// Mitsubishi GX Works2 project: 乙級第三題-ST   PLC: FX3U/FX3UC

// task Task_01 (event TRUE, interval 0, priority 31): POU_01

PROGRAM POU_01
VAR
  wProgramStep : INT;
  wPulse : INT;
  wSpeed : INT;
  tdT143 : TON;
  tdT201 : TON;
  tdT202 : TON;
  bM0 : BOOL;
  bServoRun : BOOL;
  bServoRev : BOOL;
  bM143 : BOOL;
  bM133 : BOOL;
  bM17 : BOOL;
  tdT200 : TON;
  tdT144 : TON;
  tdT203 : TON;
  bStarted : BOOL;
  tdTX11 : TON;
  trigX11 : F_TRIG;
  tdT50 : TON;
  tdT21 : TON;
  tdT60 : TON;
  tdT61 : TON;
  tdT70 : TON;
  tdT73 : TON;
  tdT62 : TON;
  tdT43 : TON;
  tdT71 : TON;
  tdT75 : TON;
  tdT42 : TON;
  tdT72 : TON;
  tdT22 : TON;
  tdT24 : TON;
  tdT27 : TON;
  tdT28 : TON;
END_VAR
VAR CONSTANT
  W_ORG_POS : INT := 16100;
  W_FRONT_INSTALL_POS : INT := 13600;
END_VAR
VAR
  tdT30 : TON;
  tdT31 : TON;
  tdT33 : TON;
  tdT35 : TON;
  tdT25 : TON;
  tdT36 : TON;
  bJawClosed : BOOL;
  bReachOrg : BOOL;
END_VAR
VAR CONSTANT
  W_REAR_INSTALL_POS : INT := 9600;
END_VAR
(* 機電整合乙級術科第三題
   Author: Steven Luo
   Date: 2018/10/25
*)

IF M8000 THEN
	Y17 := TRUE;
END_IF;

IF M8002 THEN
	D8342 := 3000;
	D8343 := 10000;
	D8348 := 1000;
	D8349 := 1000;
	bServoRun := FALSE;
	bServoRev := FALSE;
	bM0 := FALSE;
	bM17 := FALSE;
	bM143 := FALSE;
	tdT200(IN := FALSE);
	wProgramStep := 0;
END_IF;

IF M133 THEN
	bM133 := TRUE;
END_IF;

IF Y11 THEN
	bJawClosed := TRUE;
ELSE
	bJawClosed := FALSE;
END_IF;

IF NOT M144 AND NOT bM17 THEN
	IF bM0 THEN
		D5 := 0;
	ELSE
		D5 := 310;
	END_IF;
END_IF;

IF NOT X17 THEN (* 急停 *)
	ZRST(TRUE, Y0, Y10);
	ZRST(TRUE, Y13, Y16);
(*	M8349 := TRUE;*)
	bServoRun := FALSE;
	D5 := 313;
	bStarted := FALSE;
	bM17 := TRUE;
	M144 := FALSE;
	tdT201(IN := FALSE);
	tdT202(IN := FALSE);
	tdT203(IN := FALSE);
	wProgramStep := -1;
END_IF;

IF X17 AND bM17 AND M136 THEN
	D5 := 312;
(*	M8349 := FALSE;*)
	IF M132 THEN (* 解除急停，按下復歸 *)
		bM17 := FALSE;
		bM143 := TRUE;
		tdT143(IN := FALSE);
		tdT144(IN := FALSE);
		wProgramStep := 201;
	END_IF;
END_IF;

IF bM143 THEN (* 黃燈閃爍 *)
	tdT143(IN := NOT tdT144.Q, PT := T#500ms);
	tdT144(IN := tdT143.Q, PT := T#500ms);
	M143 := tdT143.Q;
END_IF;

IF X3 AND X6 AND NOT Y13 AND NOT Y14 AND NOT Y15 AND NOT Y16 AND NOT M136 THEN
	IF D8140 = W_ORG_POS THEN 
		bM0 := TRUE; (* 原點條件 *)
	END_IF;
ELSE
	bM0 := FALSE;
END_IF;

PLSR(bServoRun, wSpeed, wPulse, D8349, Y0);
OUT(bServoRev, Y4);

D4 := D1 + D2 + D3;

CASE wProgramStep OF
0:
	IF X17 THEN
		IF M130 THEN
			tdT201(IN := FALSE);
			tdT202(IN := FALSE);
			tdT203(IN := FALSE);
			wProgramStep := 200;
		ELSE
			wProgramStep := 20;
		END_IF;
	END_IF;
20:
	IF M130 THEN
		wProgramStep := 0;
	END_IF;
	IF bM0 THEN
		ZRST(TRUE, D0, D5);
		ZRST(TRUE, M150, M152);
		ZRST(TRUE, M160, M164);
		bM133 := FALSE;
		bM143 := FALSE;
		bReachOrg := FALSE;
		M142 := TRUE;
		M143 := FALSE;
		M144 := FALSE;
		tdT21(IN := FALSE);
		tdT22(IN := FALSE);
		tdT24(IN := FALSE);
		tdT25(IN := FALSE);
		tdT27(IN := FALSE);
		tdT28(IN := FALSE);
		tdT30(IN := FALSE);
		tdT31(IN := FALSE);
		tdT33(IN := FALSE);
		tdT35(IN := FALSE);
		tdT36(IN := FALSE);
		tdT42(IN := FALSE);
		tdT43(IN := FALSE);
		tdT50(IN := FALSE);
		tdT60(IN := FALSE);
		tdT61(IN := FALSE);
		tdT62(IN := FALSE);
		tdT70(IN := FALSE);
		tdT71(IN := FALSE);
		tdT72(IN := FALSE);
		tdT73(IN := FALSE);
		tdT75(IN := FALSE);
		tdTX11(IN := FALSE);
		IF M131 THEN
			bStarted := TRUE;
			M142 := FALSE;
			M144 := TRUE;
			wProgramStep := 21;
		END_IF;
	END_IF;
21:
	Y14 := TRUE; (* F輸送帶運轉 *)
	Y15 := TRUE; (* 定位缸 *)
	tdT21(IN := TRUE, PT := T#3s);
	IF tdT21.Q THEN
		Y14 := FALSE;
		Y15 := FALSE;
		wProgramStep := 20;
	END_IF;
	tdTX11(IN := TRUE, PT := T#2s);
	IF X11 THEN
		D20 := TIME_TO_INT(tdTX11.ET);
		ZCP(TRUE, 900, 1300, TIME_TO_INT(tdTX11.ET), M150);
		INCP(TRUE, D0);
	END_IF;
	trigX11(_CLK := X11);
	IF trigX11.Q THEN
		IF M150 THEN (* 凹槽朝前 *)
			wProgramStep := 60;
		ELSIF M151 THEN (* 凹槽朝後 *)
			wProgramStep := 60;
		ELSIF M152 THEN (* 凹槽朝下 *)
			wProgramStep := 50;
		END_IF;
	END_IF;
22: (* 組裝料組裝行程 *)
	Y15 := FALSE; (* 進料缸 *)
	Y6 := TRUE; (* B-水平缸縮回 *)
	IF X3 THEN (* Y軸氣壓缸後位 *)
		Y6 := FALSE;
		wProgramStep := 23;
	END_IF;
23:
	Y7 := TRUE; (* C+垂直缸下降 *)
	IF X7 THEN (* Z軸氣壓缸下位 *)
		Y7 := FALSE;
		wProgramStep := 24;
	END_IF;
24:
	tdT24(IN := TRUE, PT := T#500ms);
	IF tdT24.Q THEN
		wProgramStep := 25;
	END_IF;
25:
	Y11 := FALSE;
	Y12 := TRUE; (* D-夾爪放 *)
	tdT25(IN := TRUE, PT := T#500ms);
	IF tdT25.Q THEN
		Y12 := FALSE;
		IF M150 THEN
			M160 := FALSE;
		ELSIF M151 THEN
			M161 := FALSE;
		END_IF;
		wProgramStep := 26;
	END_IF;
26:
	Y10 := TRUE; (* C-垂直缸上升 *)
	IF X6 THEN (* Z軸氣壓缸上位 *)
		Y10 := FALSE;
		wProgramStep := 27;
	END_IF;
27:
	Y13 := TRUE; (* E分離缸分離 *)
	tdT27(IN := TRUE, PT := T#1000ms);
	IF tdT27.Q THEN
		Y13 := FALSE;
		wProgramStep := 28;
	END_IF;
28:
	IF X10 THEN
		D5 := 310;
		wPulse := W_FRONT_INSTALL_POS;
		bServoRun := TRUE;
		bServoRev := TRUE;
		tdT28(IN := TRUE, PT := T#500ms);
		IF NOT M8340 AND tdT28.Q THEN
			bServoRun := FALSE;
			bServoRev := FALSE;
			wProgramStep := 29;
		END_IF;
	ELSE
		D5 := 311;
	END_IF;
29:
	Y7 := TRUE; (* C+垂直缸下降 *)
	IF X7 THEN (* Z軸氣壓缸下位 *)
		Y7 := FALSE;
		wProgramStep := 30;
	END_IF;
30:
	tdT30(IN := TRUE, PT := T#500ms);
	IF tdT30.Q THEN
		wProgramStep := 31;
	END_IF;
31:
	Y11 := TRUE; (* D+夾爪夾 *)
	tdT31(IN := TRUE, PT := T#500ms);
	IF tdT31.Q THEN
		M162 := TRUE; (* 圓料夾取 *)
		wProgramStep := 32;
	END_IF;
32:
	Y10 := TRUE; (* C-垂直缸上升 *)
	IF X6 THEN (* Z軸氣壓缸上位 *)
		Y10 := FALSE;
		wProgramStep := 33;
	END_IF;
33:
	wPulse := W_FRONT_INSTALL_POS;
	bServoRun := TRUE;
	tdT33(IN := TRUE, PT := T#500ms);
	IF NOT M8340 AND tdT33.Q THEN
		bServoRun := FALSE;
		wProgramStep := 34;
	END_IF;
34:
	Y7 := TRUE; (* C+垂直缸下降 *)
	IF X7 THEN (* Z軸氣壓缸下位 *)
		Y7 := FALSE;
		wProgramStep := 35;
	END_IF;
35:
	Y11 := FALSE;
	Y12 := TRUE; (* D-夾爪放 *)
	tdT35(IN := TRUE, PT := T#500ms);
	IF tdT35.Q THEN
		Y12 := FALSE;
		M162 := FALSE;
		wProgramStep := 36;
	END_IF;
36:
	Y11 := TRUE; (* D+夾爪夾 *)
	tdT36(IN := TRUE, PT := T#500ms);
	IF tdT36.Q THEN
		IF M150 THEN
			M163 := TRUE; (* 凹槽朝前組裝 *)
		ELSIF M151 THEN
			M164 := TRUE; (* 凹槽朝後組裝 *)
		END_IF;
		wProgramStep := 37;
	END_IF;
37: (* 組裝料出料行程 *)
	Y10 := TRUE; (* C-垂直缸上升 *)
	IF X6 THEN (* Z軸氣壓缸上位 *)
		Y10 := FALSE;
		D1 := D1 + 1;
		wProgramStep := 70;
	END_IF;
40:
	Y5 := TRUE; (* B+水平缸伸出 *)
	IF X5 THEN (* Y軸氣壓缸前位 *)
		Y5 := FALSE;
		wProgramStep := 41;
	END_IF;
41:
	Y7 := TRUE; (* C+垂直缸下降 *)
	IF X7 THEN (* Z軸氣壓缸下位 *)
		Y7 := FALSE;
		wProgramStep := 42;
	END_IF;
42:
	tdT42(IN := TRUE, PT := T#500ms);
	IF tdT42.Q THEN
		wProgramStep := 43;
	END_IF;
43:
	Y11 := TRUE; (* D+夾爪夾 *)
	tdT43(IN := TRUE, PT := T#500ms);
	IF tdT43.Q THEN
		IF M150 THEN
			M160 := TRUE;
		ELSIF M151 THEN
			M161 := TRUE;
		END_IF;
		wProgramStep := 44;
	END_IF;
44:
	Y10 := TRUE; (* C-垂直缸上升 *)
	IF X6 THEN (* Z軸氣壓缸上位 *)
		Y10 := FALSE;
		IF M150 THEN
			wProgramStep := 22;
		ELSE
			wProgramStep := 45;
		END_IF;
	END_IF;
45: (* 非組裝料出料行程 *)
	Y6 := TRUE; (* B-水平缸縮回 *)
	IF X4 THEN (* Y軸氣壓缸中位 *)
		Y6 := FALSE;
		D2 := D2 + 1;;
		wProgramStep := 70;
	END_IF;
50: (* 反面出料行程 *)
	Y16 := TRUE; (* H定位缸 *)
	tdT50(IN := TRUE, PT := T#2500ms);
	IF tdT50.Q THEN
		Y16 := FALSE;
		D3 := D3 + 1;
		wProgramStep := 60;
	END_IF;
60:
	tdT60(IN := TRUE, PT := T#2500ms);
	IF tdT60.Q THEN
		Y14 := FALSE; (* F輸送帶停止 *)
		IF M150 THEN
			wProgramStep := 40;
		ELSE
			wProgramStep := 61;
		END_IF;
	END_IF;
61:
	tdT61(IN := TRUE, PT := T#500ms);
	IF tdT61.Q THEN
		wProgramStep := 62;
	END_IF;
62:
	Y15 := FALSE; (* 進料缸 *)
	tdT62(IN := TRUE, PT := T#500ms);
	IF tdT62.Q THEN
		IF M151 THEN
			wProgramStep := 40;
		ELSE
			IF NOT bM133 THEN
				tdT21(IN := FALSE);
				tdT22(IN := FALSE);
				tdT24(IN := FALSE);
				tdT25(IN := FALSE);
				tdT27(IN := FALSE);
				tdT28(IN := FALSE);
				tdT30(IN := FALSE);
				tdT31(IN := FALSE);
				tdT33(IN := FALSE);
				tdT35(IN := FALSE);
				tdT36(IN := FALSE);
				tdT42(IN := FALSE);
				tdT43(IN := FALSE);
				tdT50(IN := FALSE);
				tdT60(IN := FALSE);
				tdT61(IN := FALSE);
				tdT62(IN := FALSE);
				tdT70(IN := FALSE);
				tdT71(IN := FALSE);
				tdT72(IN := FALSE);
				tdT73(IN := FALSE);
				tdT75(IN := FALSE);
				tdTX11(IN := FALSE);
				wProgramStep := 21;
			ELSE
				wProgramStep := 0;
			END_IF;
		END_IF;
	END_IF;
70: (* 排料 *)
	wPulse := W_ORG_POS;
	wSpeed := D8343;
	bServoRun := TRUE;
	tdT70(IN := TRUE, PT := T#500ms);
	IF NOT M8340 AND tdT70.Q THEN
		bServoRun := FALSE;
		bReachOrg := TRUE;
		D8140 := 0;
		Y3 := TRUE; (* Servo CCLR *)
		tdT71(IN := TRUE, PT := T#500ms);
		IF tdT71.Q THEN
			Y3 := FALSE;
			wProgramStep := 71;
		END_IF;
	END_IF;
71:
	Y7 := TRUE; (* C+垂直缸下降 *)
	IF X7 THEN (* Z軸氣壓缸下位 *)
		Y7 := FALSE;
		IF M162 THEN
			wProgramStep := 73;
		ELSE
			wProgramStep := 72;
		END_IF;
	END_IF;
72:
	tdT72(IN := TRUE, PT := T#500ms);
	IF tdT72.Q THEN
		wProgramStep := 73;
	END_IF;
73:
	Y11 := FALSE;
	Y12 := TRUE; (* D-夾爪放 *)
	tdT73(IN := TRUE, PT := T#500ms);
	IF tdT73.Q THEN
		Y12 := FALSE;
		wProgramStep := 74;
	END_IF;
74:
	Y10 := TRUE; (* C-垂直缸上升 *)
	IF X6 THEN (* Z軸氣壓缸上位 *)
		Y10 := FALSE;
		wProgramStep := 75;
	END_IF;
75:
	wPulse := W_ORG_POS;
	bServoRun := TRUE;
	bServoRev := TRUE;
	tdT75(IN := TRUE, PT := T#500ms);
	IF NOT M8340 AND tdT75.Q THEN
		bServoRun := FALSE;
		bServoRev := FALSE;
		wProgramStep := 76;
	END_IF;
76:
	Y6 := TRUE; (* B-水平缸縮回 *)
	IF X3 THEN (* Y軸氣壓缸後位 *)
		Y6 := FALSE;
		IF NOT bM133 AND NOT bM143 THEN
			tdT21(IN := FALSE);
			tdT22(IN := FALSE);
			tdT24(IN := FALSE);
			tdT25(IN := FALSE);
			tdT27(IN := FALSE);
			tdT28(IN := FALSE);
			tdT30(IN := FALSE);
			tdT31(IN := FALSE);
			tdT33(IN := FALSE);
			tdT35(IN := FALSE);
			tdT36(IN := FALSE);
			tdT42(IN := FALSE);
			tdT43(IN := FALSE);
			tdT50(IN := FALSE);
			tdT60(IN := FALSE);
			tdT61(IN := FALSE);
			tdT62(IN := FALSE);
			tdT70(IN := FALSE);
			tdT71(IN := FALSE);
			tdT72(IN := FALSE);
			tdT73(IN := FALSE);
			tdT75(IN := FALSE);
			tdTX11(IN := FALSE);
			wProgramStep := 21;
		ELSE
			wProgramStep := 0;
		END_IF;
	END_IF;
100:
	Y5 := TRUE; (* B+水平缸伸出 *)
	IF X5 THEN (* Y軸氣壓缸前位 *)
		Y5 := FALSE;
		wProgramStep := 71;
	END_IF;
101:
	Y6 := TRUE; (* B-水平缸縮回 *)
	IF X3 THEN (* Y軸氣壓缸後位 *)
		Y6 := FALSE;
		wProgramStep := 102;
	END_IF;
102:
	Y5 := TRUE; (* B+水平缸伸出 *)
	IF X4 THEN (* Y軸氣壓缸中位 *)
		Y5 := FALSE;
		wProgramStep := 71;
	END_IF;
200:
	IF X6 THEN (* c0 Z軸上位 *)
		IF X3 THEN (* b0 Y軸後位 *)
			wSpeed := D8343;
			wPulse := 3000;
			OUT((NOT X0 AND M110) OR M111, bServoRun);
			OUT(M111 AND NOT M110, bServoRev);
			IF X0 THEN
				D8140 := 0;
				Y3 := TRUE; (* Servo CCLR *)
				tdT200(IN := TRUE, PT := T#500ms);
				IF tdT200.Q THEN
					Y3 := FALSE;
				END_IF;
			ELSE
				tdT200(IN := FALSE);
			END_IF;
		END_IF;
		OUT(M112, Y5); (* B+水平缸伸出 *)
		OUT(M113, Y6); (* B-水平缸縮回 *)
	END_IF;
	OUT(M114, Y10); (* C-垂直缸上升 *)
	OUT(M115, Y7); (* C+垂直缸下降 *)
	OUT(M116, Y11); (* D+夾爪夾 *)
	OUT(M117, Y12); (* D-夾爪放 *)
	OUT(M119, Y14); (* F輸送帶運轉 *)
	OUT(M118, Y13); (* E分離缸分離 *)
	OUT(M120, Y15); (* G進料缸進料 *)
	OUT(M121, Y16); (* H定位缸 *)
	IF M137 OR M132 THEN (* servo hoome *)
		wProgramStep := 201;
	END_IF;
	IF NOT M130 THEN
		wProgramStep := 0;
	END_IF;
201:
	Y10 := TRUE; (* C-垂直缸上升 *)
	IF X6 THEN
		Y10 := FALSE;
		Y6 := TRUE; (* B-水平缸縮回 *)
		IF X3 THEN
			Y6 := FALSE;
			IF bReachOrg THEN
				wProgramStep := 202;
			ELSE
				wPulse := 32767;
				wSpeed := D8343;
				OUT(NOT X0, bServoRun);
				IF X0 THEN
					wProgramStep := 202;
				END_IF;
			END_IF;
		END_IF;
	END_IF;
202:
	IF NOT bReachOrg THEN
		wPulse := 1000;
		wSpeed := 1000;
		bServoRun := TRUE;
	END_IF;
	tdT201(IN := TRUE, PT := T#500ms);
	IF NOT M8340 AND tdT201.Q THEN
		bServoRun := FALSE;
		D8140 := 0;
		Y3 := TRUE; (* Servo CCLR *)
		tdT202(IN := TRUE, PT := T#500ms);
		IF tdT202.Q THEN
			wSpeed := D8343;
			Y3 := FALSE;
			IF M160 THEN
				wProgramStep := 71;
			ELSIF M161 THEN
				wProgramStep := 101;
			ELSIF M163 OR M164 THEN
				wProgramStep := 71;
			ELSIF M162 THEN
				wProgramStep := 100;
			ELSE
				wProgramStep := 203;
			END_IF;
		END_IF;
	END_IF;
203:
	wPulse := W_ORG_POS;
	bServoRun := TRUE;
	bServoRev := TRUE;
	tdT203(IN := TRUE, PT := T#500ms);
	IF NOT M8340 AND tdT203.Q THEN
		bServoRun := FALSE;
		bServoRev := FALSE;
		wProgramStep := 0;
	END_IF;
END_CASE;
END_PROGRAM
